// TIA Portal V20 export
// export: Created 2025-12-01T14:57:21.0471839Z, ExportSetting None, DisplayName Totally Integrated Automation Portal, DisplayVersion V20 Update 3, DisplayName TIA Portal Openness, DisplayVersion V20 Update 3, DisplayName TIA Portal Version Control Interface, DisplayVersion V20 Update 3, DisplayName STEP 7 Professional, DisplayVersion V20 Update 3, DisplayName STEP 7 Safety, DisplayVersion V20 Update 2, DisplayName WinCC Basic/Comfort/Advanced, DisplayVersion V20 Update 3, DisplayName WinCC Professional, DisplayVersion V20 Update 3, DisplayName WinCC Unified, DisplayVersion V20 Update 3
DATA_BLOCK "DB2125_DB_LinPot_Maq1"   // DB2125, F_DB
FAMILY : FPRI0855
VERSION : 0.0
// stored: AutoNumber false, InstanceOfName FB2133_F_LinPot_Maquina, InstanceOfType FB
"FB2133_F_LinPot_Maquina"
   // VAR_INPUT
   //    NumArmario : Int;
   //    NumLinea : Int;
   //    Maquina_OFF : Bool;
   //    Proteccion : Bool;
   //    Seguridades : Bool;
   //    FEEDBACK : Bool;
   //    Rearme : Bool;
   //    QBAD_FIO : Bool;
   //    FDB_TIME : Time;
   // END_VAR
   // VAR_OUTPUT
   //    Q : Bool;
   //    ERROR : Bool;
   //    H : Bool;
   // END_VAR
   // VAR
   //    F_FDBACK { S7_SetPoint := 'True'} : FDBACK;
   //    F_ESTOP1 { S7_SetPoint := 'True'} : ESTOP1;
   // END_VAR
BEGIN
END_DATA_BLOCK
